FUNCTION_BLOCK MotionAxisO
VAR
	(* Axis Reference *)
	axisRef : AXIS_REF; 
	
	(* Motion Function Block *)
	fbMcPower 		: MC_Power;				// FB for enable and override
	fbMcReset 		: MC_Reset;				// FB to reset axis
	fbMcStop 		: MC_Stop;				// FB to stop axis
	fbMcHalt		: MC_Halt;				// FB to halt axis
	fbMcMoveAbsolute: MC_MoveAbsolute;		// FB to move axis (Absolute Move)
	fbMcMoveRelative: MC_MoveRelative;		// FB to move axis (Relative Move)
	fbMcJog         : MC_Jog;				// FB to move axis (Relative Move)
	
	(* Axis Config Settings *)
	axisConfig : AxisConfigurationO;
	
	(* Axis Status *)
	axisStatus : BOOL;
	blockError : BOOL;
	nErrorID	   : UDINT;

END_VAR

METHOD AbsoluteMove : BOOL
VAR_INPUT
	TargetPosition : LREAL;
END_VAR

VAR
END_VAR
END_METHOD

PROPERTY ActualPosition : LReal
GET
ActualPosition := axisRef.NcToPlc.ActPos;
END_GET
END_PROPERTY

PROPERTY ActualSpeed : LReal
GET
ActualSpeed := axisRef.NcToPlc.ActVelo;
END_GET
END_PROPERTY

PROPERTY AxisState : BOOL
GET
AxisState:= axisRef.NcToPlc.StateDWord.0 AND axisStatus ;
END_GET
END_PROPERTY

METHOD configure :BOOL;
VAR_INPUT
	stAxisConfig : AxisConfigurationO;
END_VAR
axisConfig := stAxisConfig;

//Not Implemented
configure:=TRUE;
END_METHOD

METHOD Disable : BOOL
VAR
END_VAR
Disable := mcPower(enable:=FALSE);
END_METHOD

METHOD Enable : BOOL
VAR
END_VAR
Enable := mcPower(enable:=TRUE);
END_METHOD

PROPERTY Error : Bool
GET
Error := axisRef.NcToPlc.StateDWord.31 OR blockError;
END_GET
END_PROPERTY

PROPERTY ErrorID : UDINT
GET
ErrorID := nErrorID;
END_GET
END_PROPERTY

METHOD Jog : BOOL;
VAR_INPUT
	JogFrw : BOOL;
	JogRev : BOOL;
END_VAR
Jog := mcJog(jogFrw:=JogFrw,jogRev:=JogRev);
END_METHOD

METHOD INTERNAL mcJog : BOOL
VAR_INPUT
	jogFrw : BOOL;
	jogRev : BOOL;
END_VAR
(* Jog Frw/Rev *)
fbMcJog(
		Axis:=axisRef, 
		JogForward:=jogFrw, 
		JogBackwards:=jogRev, 
		Mode:=axisConfig.JogMode, 
		Position:=axisConfig.JogInchingPosition, 
		Velocity:=axisConfig.JogVelocity, 
		Acceleration:=axisConfig.JogAccleration, 
		Deceleration:=axisConfig.JogDeaccleration);
		
(* Error Handling *)
IF fbMcJog.Error THEN
	blockError:= TRUE;
	nErrorID := fbMcJog.ErrorID;
END_IF

(* Jog State *)
mcJog := fbMcJog.Active;
END_METHOD

METHOD mcMoveAbs : BOOL
VAR_INPUT
	TargetPosition : LREAL;
END_VAR

VAR
	previousTargetPosition : LREAL;
END_VAR
(* Absloute Move *)
IF TargetPosition <> previousTargetPosition THEN
	
END_IF

(* Absloute Move Block *)
fbMcMoveAbsolute(
				Axis:= axisRef, 
				Execute:= , 
				Position:= , 
				Velocity:= , 
				Acceleration:= , 
				Deceleration:= , 
				Jerk:= , 
				BufferMode:= , 
				Options:= , 
				Done=> , 
				Busy=> , 
				Active=> , 
				CommandAborted=> , 
				Error=> , 
				ErrorID=> );
		
(* Error Handling *)
IF fbMcMoveAbsolute.Error THEN
	blockError:= TRUE;
	nErrorID := fbMcMoveAbsolute.ErrorID;
END_IF

(* Absolute Move Complete *)
mcMoveAbs := fbMcMoveAbsolute.Done AND NOT fbMcMoveAbsolute.Busy ;
END_METHOD

METHOD INTERNAL mcPower : BOOL
VAR_INPUT
	enable : BOOL;
END_VAR
(* Axis Enable/Disable *)
fbMCPower(Enable 			:= enable, 
		  Enable_Positive	:= axisConfig.EnablePositive, 
		  Enable_Negative	:= axisConfig.EnableNegative, 
		  Override		    := axisConfig.Override,
	      Axis			    := axisRef);

(* Error Handling *)
IF fbMcPower.Error THEN
	blockError:= TRUE;
	nErrorID := fbMcPower.ErrorID;
END_IF

(* Axis State *)
mcPower := axisStatus := fbMCPower.Status;
END_METHOD

END_FUNCTION_BLOCK

(* stored: Version 1.1.0.1, ProductVersion 3.1.4024.12
   POU MotionAxisO: Id {6efac28a-a867-4ac1-8d79-383fd5b163f6}, SpecialFunc None
   Method AbsoluteMove: Id {c3451ace-de85-4b3d-85a3-1bb2311490ba}
   Property ActualPosition: Id {b53e2779-5fd6-4938-833e-613ccdf9545b}
   Get Get: Id {186b8ccb-2b3b-4cae-8cee-7170028d065c}
   Property ActualSpeed: Id {a120a2d9-432c-4e75-ae40-182a022fe029}
   Get Get: Id {3de0044e-9dac-4dce-a533-695a02650e46}
   Property AxisState: Id {dee10592-fb1a-458c-b8d9-450e0e9a9721}
   Get Get: Id {a4ce2992-626b-43c0-9473-a8c49978d3ed}
   Method configure: Id {05b83e6f-6c9d-482c-87c5-d51b21ad4cdc}
   Method Disable: Id {cdc7a590-792f-495b-82e0-a680f5fc044e}
   Method Enable: Id {b3550f0a-fa67-4c80-947d-d090edf7c896}
   Property Error: Id {557a2853-1fb5-40b5-8793-ea3e16bdc4b0}
   Get Get: Id {1686439e-d75c-4357-bde7-a1f797103e23}
   Property ErrorID: Id {dcfddad3-85dc-4a25-b1e7-e9c8b2439f63}
   Get Get: Id {974c0fe1-5ff3-4882-9d23-7536fa5d4618}
   Method Jog: Id {6cea3643-adb1-4590-ade4-876e97b45011}
   Method mcJog: Id {67145e7d-43ee-4162-be9f-bb2cfc9fa1ce}
   Method mcMoveAbs: Id {53fe8ef5-1ece-4d4f-9cac-020d395096eb}
   Method mcPower: Id {09f11a1e-6091-410a-b73b-ed1a52c5c7e7} *)
